// TIA Portal project "Servomotor" (V20)

(* hardware
DEVICE "S7-1500/ET200MP-Station_1"  S7-1500 station
   slot 0: "Profilschiene_0"  Rack  6ES7 590-1***0-0AA0
   slot 1: "PLC_1"  CPU 1515-2 PN  6ES7 515-2AM02-0AB0  V2.9
      slot 3: "CPU-Display_1"  6ES7591-1BA00-0AA0
      slot 32768: "PROFINET-Schnittstelle_1"  X1
         slot 32769: "Port_1"  X1 P1
         slot 32770: "Port_2"  X1 P2
      slot 33024: "PROFINET-Schnittstelle_2"  X2
         slot 33025: "Port_1"  X2 P1
      slot 34817: "Virtual CP interface port_1"  Virtual CP interface port  Virtual CP interface port
   slot 2: "AQ 8xU/I HS_1"  AQ 8xU/I HS  6ES7 532-5HF00-0AB0  V2.2
DEVICE "SINAMICS S_1"  SINAMICS S210
   slot 0: "Antriebsgerät_X"  S210 PN  6SL3210-5HB10-4xFx  V5.2.3
      slot 1: "PROFINET-Schnittstelle"  PROFINET
      slot 3: "Ethernet-IBN-Schnittstelle"  LAN
   slot 0: "Antriebsregelung"  S210 PN
      slot 200: "Power Module_1"  Antriebsregelung  6SL3210-5HB10-4xFx
      slot 300: "Geberauswertung_1"  Antriebsregelung  1FK2103-4AG0x-xDxx
      slot 400: "Messsystem_1"  Antriebsregelung  1FK2103-4AG0x-xDxx
      slot 1000: "Motor_1"  Antriebsregelung  1FK2103-4AG0x-xDxx
DEVICE "SINAMICS S_2"  SINAMICS S210
   slot 0: "Antriebsgerät_Y"  S210 PN  6SL3210-5HB10-4xFx  V5.2.3
      slot 1: "PROFINET-Schnittstelle"  PROFINET
      slot 3: "Ethernet-IBN-Schnittstelle"  LAN
   slot 0: "Antriebsregelung"  S210 PN
      slot 200: "Power Module_1"  Antriebsregelung  6SL3210-5HB10-4xFx
      slot 300: "Geberauswertung_1"  Antriebsregelung  1FK2103-4AG0x-xDxx
      slot 400: "Messsystem_1"  Antriebsregelung  1FK2103-4AG0x-xDxx
      slot 1000: "Motor_1"  Antriebsregelung  1FK2103-4AG0x-xDxx
DEVICE "SCALANCE X-200 IRT"  SCALANCE X-Station
   slot 0: "SCALANCE X-Rack"  Rail
   slot 0: "Switch_1"  SCALANCE X204 IRT  6GK5 204-0BA00-2BA3  V5.6
*)

// ===== PLC "PLC_1"  CPU 1515-2 PN =====

VAR_GLOBAL   // PLC tag table "Standard-Variablentabelle"
   "Tag_1" AT %AW30 : Int;
   "Tag_2" AT %AW32 : Int;
END_VAR

TYPE "typePOS_Axis"
   STRUCT
      Taster : Struct
         Power : Bool;
         Reset : Bool;
         Home : Bool;
         Halt : Bool;
         MoveAbsolute : Bool;
         MoveRelative : Bool;
         MoveVelocity : Bool;
         MoveJogForward : Bool;
         MoveJogBackward : Bool;
         Stop : Bool;
      END_STRUCT;
      Eingaben : Struct
         Absolutposition : LReal;
         Relativbewegung : LReal;
         Geschwindigkeit : LReal;
      END_STRUCT;
      Anzeigen : Struct
         TO_freigegeben : Bool;
         TO_referenziert : Bool;
         Sammelfehler : Bool;
         Done : Struct
            Power : Bool;
            Reset : Bool;
            Home : Bool;
            Halt : Bool;
            MoveAbsolute : Bool;
            MoveRelative : Bool;
            MoveVelocity : Bool;
            MoveJog : Bool;
            Stop : Bool;
         END_STRUCT;
         Busy : Struct
            Power : Bool;
            Reset : Bool;
            Home : Bool;
            Halt : Bool;
            MoveAbsolute : Bool;
            MoveRelative : Bool;
            MoveVelocity : Bool;
            MoveJog : Bool;
            Stop : Bool;
         END_STRUCT;
         CommandAborted : Struct
            Power : Bool;
            Reset : Bool;
            Home : Bool;
            Halt : Bool;
            MoveAbsolute : Bool;
            MoveRelative : Bool;
            MoveVelocity : Bool;
            MoveJog : Bool;
            Stop : Bool;
         END_STRUCT;
         Fehler : Struct
            Power : Bool;
            Reset : Bool;
            Home : Bool;
            Halt : Bool;
            MoveAbsolute : Bool;
            MoveRelative : Bool;
            MoveVelocity : Bool;
            MoveJog : Bool;
            Stop : Bool;
         END_STRUCT;
         Error_ID : Struct
            Power : Word;
            Reset : Word;
            Home : Word;
            Halt : Word;
            MoveAbsolute : Word;
            MoveRelative : Word;
            MoveVelocity : Word;
            MoveJog : Word;
            Stop : Word;
         END_STRUCT;
      END_STRUCT;
      Ausgaben : Struct
         Position : LReal;
         ActualPosition : LReal;
         ActualVelocity : LReal;
         ActualAcceleration : LReal;
      END_STRUCT;
   END_STRUCT;
END_TYPE

DATA_BLOCK "Daten"   // DB100
{ S7_Optimized_Access := 'TRUE' }
VERSION : 0.1
   VAR
      Daten_X_Achse : "typePOS_Axis";
      Daten_Y_Achse : "typePOS_Axis";
   END_VAR
BEGIN
END_DATA_BLOCK

DATA_BLOCK "IDB_Achse_X"   // DB101
{ S7_Optimized_Access := 'TRUE' }
VERSION : 0.1
// stored: InstanceOfName Achsensteuerung
"Achsensteuerung"
BEGIN
END_DATA_BLOCK

DATA_BLOCK "IDB_Achse_Y"   // DB102
{ S7_Optimized_Access := 'TRUE' }
VERSION : 0.1
// stored: InstanceOfName Achsensteuerung
"Achsensteuerung"
BEGIN
END_DATA_BLOCK

DATA_BLOCK "PositioningAxis_X"   // DB1, Motion_DB
{ S7_Optimized_Access := 'TRUE' }
AUTHOR : SIMATIC
FAMILY : MC_1500
VERSION : 6.0
// stored: InstanceOfName TO_PositioningAxis
"TO_PositioningAxis"
BEGIN
END_DATA_BLOCK

DATA_BLOCK "PositioningAxis_Y"   // DB2, Motion_DB
{ S7_Optimized_Access := 'TRUE' }
AUTHOR : SIMATIC
FAMILY : MC_1500
VERSION : 6.0
// stored: InstanceOfName TO_PositioningAxis
"TO_PositioningAxis"
BEGIN
END_DATA_BLOCK

FUNCTION_BLOCK "Achsensteuerung"   // FB101, FBD
{ S7_Optimized_Access := 'TRUE' }
VERSION : 0.1
   VAR_INPUT
      Achse : TO_PositioningAxis;
   END_VAR
   VAR_IN_OUT
      ioPOS_Axis : "typePOS_Axis";
   END_VAR
   VAR
      MDB_MC_POWER : MC_POWER;
      MDB_MC_RESET : MC_RESET;
      MDB_MC_MOVEABSOLUTE : MC_MOVEABSOLUTE;
      MDB_MC_HOME : MC_HOME;
      MDB_MC_HALT : MC_HALT;
      MD_MC_MOVERELATIVE : MC_MOVERELATIVE;
      MDB_MC_MOVEJOG : MC_MOVEJOG;
      MDB_MC_STOP : MC_STOP;
   END_VAR
BEGIN

REGION Network 1
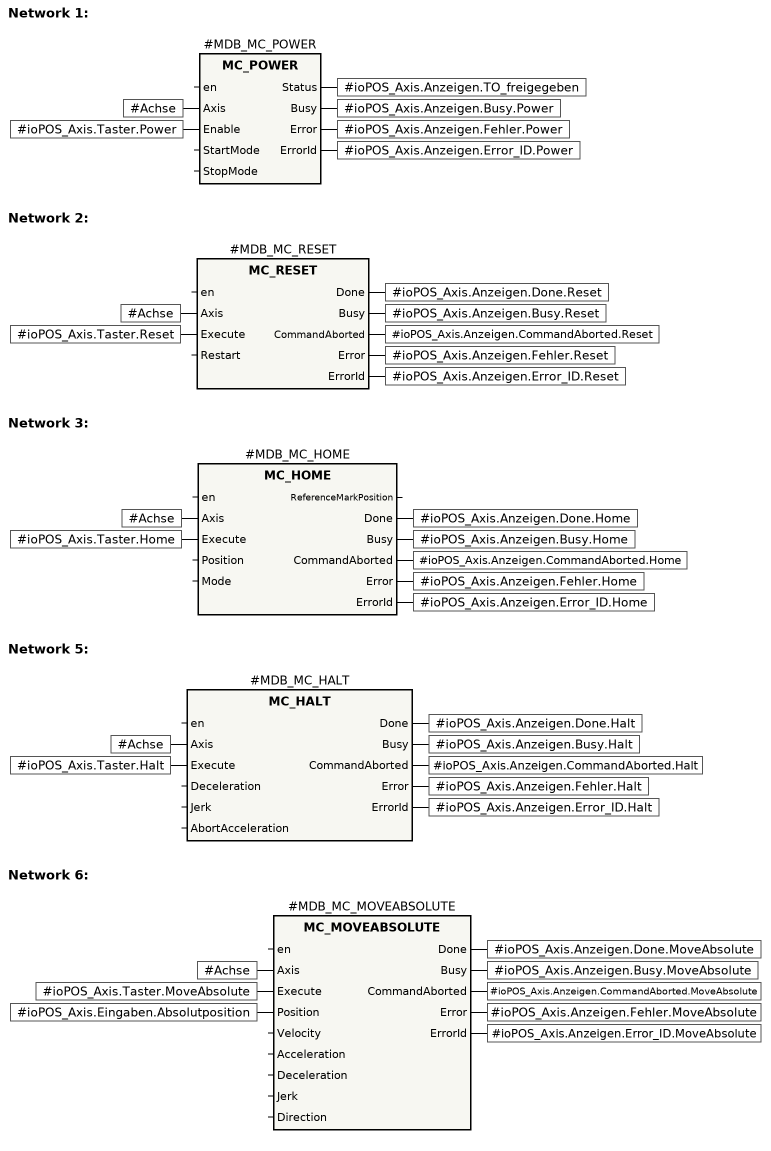
   #MDB_MC_POWER(Axis := #Achse,   // MC_POWER
                 Enable := #ioPOS_Axis.Taster.Power,
                 Status => #ioPOS_Axis.Anzeigen.TO_freigegeben,
                 Busy => #ioPOS_Axis.Anzeigen.Busy.Power,
                 Error => #ioPOS_Axis.Anzeigen.Fehler.Power,
                 ErrorId => #ioPOS_Axis.Anzeigen.Error_ID.Power);
END_REGION

REGION Network 2
   #MDB_MC_RESET(Axis := #Achse,   // MC_RESET
                 Execute := #ioPOS_Axis.Taster.Reset,
                 Done => #ioPOS_Axis.Anzeigen.Done.Reset,
                 Busy => #ioPOS_Axis.Anzeigen.Busy.Reset,
                 CommandAborted => #ioPOS_Axis.Anzeigen.CommandAborted.Reset,
                 Error => #ioPOS_Axis.Anzeigen.Fehler.Reset,
                 ErrorId => #ioPOS_Axis.Anzeigen.Error_ID.Reset);
END_REGION

REGION Network 3
   #MDB_MC_HOME(Axis := #Achse,   // MC_HOME
                Execute := #ioPOS_Axis.Taster.Home,
                Done => #ioPOS_Axis.Anzeigen.Done.Home,
                Busy => #ioPOS_Axis.Anzeigen.Busy.Home,
                CommandAborted => #ioPOS_Axis.Anzeigen.CommandAborted.Home,
                Error => #ioPOS_Axis.Anzeigen.Fehler.Home,
                ErrorId => #ioPOS_Axis.Anzeigen.Error_ID.Home);
END_REGION

REGION Network 4 (SCL)
   IF #ioPOS_Axis.Taster.Home
       AND #ioPOS_Axis.Anzeigen.Done.Home
       AND NOT #ioPOS_Axis.Anzeigen.Fehler.Home
   THEN
       #ioPOS_Axis.Anzeigen.TO_referenziert := TRUE;
   END_IF;
END_REGION

REGION Network 5
   #MDB_MC_HALT(Axis := #Achse,   // MC_HALT
                Execute := #ioPOS_Axis.Taster.Halt,
                Done => #ioPOS_Axis.Anzeigen.Done.Halt,
                Busy => #ioPOS_Axis.Anzeigen.Busy.Halt,
                CommandAborted => #ioPOS_Axis.Anzeigen.CommandAborted.Halt,
                Error => #ioPOS_Axis.Anzeigen.Fehler.Halt,
                ErrorId => #ioPOS_Axis.Anzeigen.Error_ID.Halt);
END_REGION

REGION Network 6
   #MDB_MC_MOVEABSOLUTE(Axis := #Achse,   // MC_MOVEABSOLUTE
                        Execute := #ioPOS_Axis.Taster.MoveAbsolute,
                        Position := #ioPOS_Axis.Eingaben.Absolutposition,
                        Done => #ioPOS_Axis.Anzeigen.Done.MoveAbsolute,
                        Busy => #ioPOS_Axis.Anzeigen.Busy.MoveAbsolute,
                        CommandAborted => #ioPOS_Axis.Anzeigen.CommandAborted.MoveAbsolute,
                        Error => #ioPOS_Axis.Anzeigen.Fehler.MoveAbsolute,
                        ErrorId => #ioPOS_Axis.Anzeigen.Error_ID.MoveAbsolute);
END_REGION

REGION Network 7 (SCL)
   #ioPOS_Axis.Ausgaben.Position := #Achse.Position;
   #ioPOS_Axis.Ausgaben.ActualPosition := #Achse.ActualPosition;
   #ioPOS_Axis.Ausgaben.ActualVelocity := #Achse.ActualVelocity;
   #ioPOS_Axis.Ausgaben.ActualAcceleration := #Achse.ActualAcceleration;
END_REGION

REGION Network 8
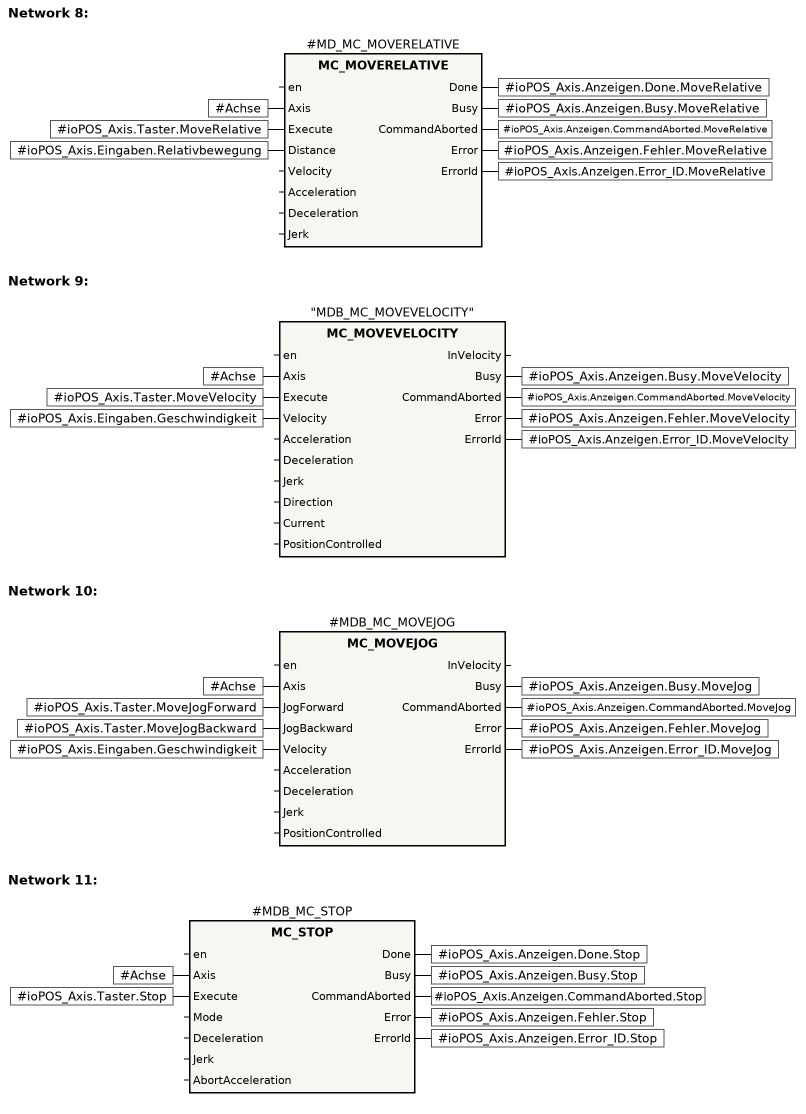
   #MD_MC_MOVERELATIVE(Axis := #Achse,   // MC_MOVERELATIVE
                       Execute := #ioPOS_Axis.Taster.MoveRelative,
                       Distance := #ioPOS_Axis.Eingaben.Relativbewegung,
                       Done => #ioPOS_Axis.Anzeigen.Done.MoveRelative,
                       Busy => #ioPOS_Axis.Anzeigen.Busy.MoveRelative,
                       CommandAborted => #ioPOS_Axis.Anzeigen.CommandAborted.MoveRelative,
                       Error => #ioPOS_Axis.Anzeigen.Fehler.MoveRelative,
                       ErrorId => #ioPOS_Axis.Anzeigen.Error_ID.MoveRelative);
END_REGION

REGION Network 9
   "MDB_MC_MOVEVELOCITY"(Axis := #Achse,   // MC_MOVEVELOCITY
                         Execute := #ioPOS_Axis.Taster.MoveVelocity,
                         Velocity := #ioPOS_Axis.Eingaben.Geschwindigkeit,
                         Busy => #ioPOS_Axis.Anzeigen.Busy.MoveVelocity,
                         CommandAborted => #ioPOS_Axis.Anzeigen.CommandAborted.MoveVelocity,
                         Error => #ioPOS_Axis.Anzeigen.Fehler.MoveVelocity,
                         ErrorId => #ioPOS_Axis.Anzeigen.Error_ID.MoveVelocity);
END_REGION

REGION Network 10
   #MDB_MC_MOVEJOG(Axis := #Achse,   // MC_MOVEJOG
                   JogForward := #ioPOS_Axis.Taster.MoveJogForward,
                   JogBackward := #ioPOS_Axis.Taster.MoveJogBackward,
                   Velocity := #ioPOS_Axis.Eingaben.Geschwindigkeit,
                   Busy => #ioPOS_Axis.Anzeigen.Busy.MoveJog,
                   CommandAborted => #ioPOS_Axis.Anzeigen.CommandAborted.MoveJog,
                   Error => #ioPOS_Axis.Anzeigen.Fehler.MoveJog,
                   ErrorId => #ioPOS_Axis.Anzeigen.Error_ID.MoveJog);
END_REGION

REGION Network 11
   #MDB_MC_STOP(Axis := #Achse,   // MC_STOP
                Execute := #ioPOS_Axis.Taster.Stop,
                Done => #ioPOS_Axis.Anzeigen.Done.Stop,
                Busy => #ioPOS_Axis.Anzeigen.Busy.Stop,
                CommandAborted => #ioPOS_Axis.Anzeigen.CommandAborted.Stop,
                Error => #ioPOS_Axis.Anzeigen.Fehler.Stop,
                ErrorId => #ioPOS_Axis.Anzeigen.Error_ID.Stop);
END_REGION

REGION Network 12 (SCL)
   // Sammelfehler
   #ioPOS_Axis.Anzeigen.Sammelfehler := #ioPOS_Axis.Anzeigen.Fehler.Power
                                       OR #ioPOS_Axis.Anzeigen.Fehler.Reset
                                       OR #ioPOS_Axis.Anzeigen.Fehler.Home
                                       OR #ioPOS_Axis.Anzeigen.Fehler.Halt
                                       OR #ioPOS_Axis.Anzeigen.Fehler.MoveAbsolute
                                       OR #ioPOS_Axis.Anzeigen.Fehler.MoveRelative
                                       OR #ioPOS_Axis.Anzeigen.Fehler.MoveVelocity
                                       OR #ioPOS_Axis.Anzeigen.Fehler.MoveJog
                                       OR #ioPOS_Axis.Anzeigen.Fehler.Stop;
END_REGION
END_FUNCTION_BLOCK

ORGANIZATION_BLOCK "Main"   // OB1, FBD, ProgramCycle
TITLE = "Main Program Sweep (Cycle)"
{ S7_Optimized_Access := 'TRUE' }
VERSION : 0.1
   VAR_INPUT
      Initial_Call : Bool;   // Initial call of this OB
      Remanence : Bool;   // =True, if remanent data are available
   END_VAR
   VAR_TEMP
      tmpNorm : LReal;
   END_VAR
BEGIN

REGION Network 1
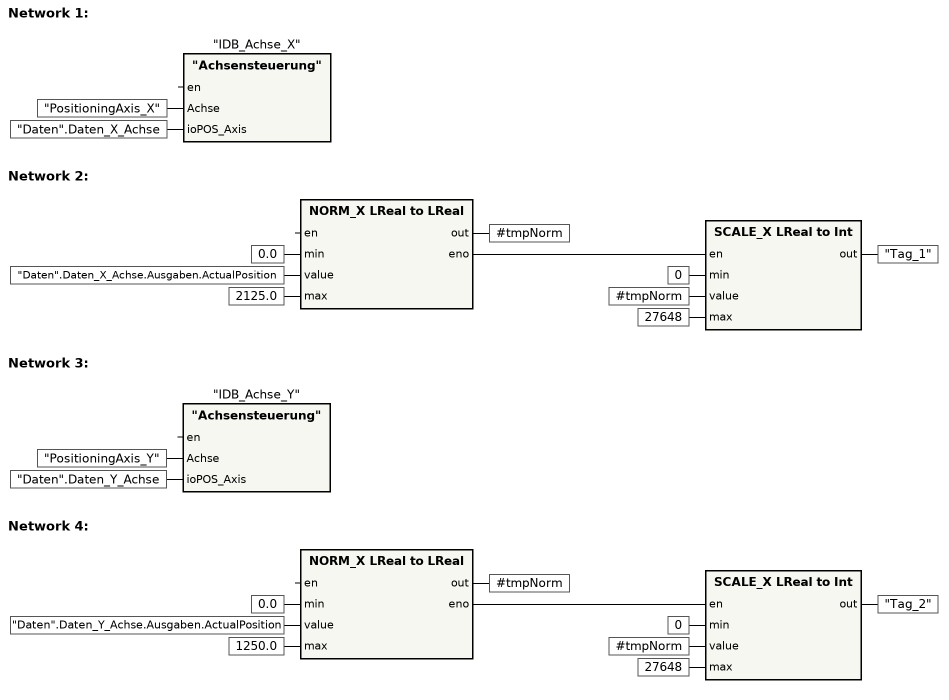
   "IDB_Achse_X"(Achse := "PositioningAxis_X", ioPOS_Axis := "Daten".Daten_X_Achse);   // "Achsensteuerung"
END_REGION

REGION Network 2
   #tmpNorm := NORM_X(MIN := 0.0, VALUE := "Daten".Daten_X_Achse.Ausgaben.ActualPosition, MAX := 2125.0);
   "Tag_1" := SCALE_X(MIN := 0, VALUE := #tmpNorm, MAX := 27648);
END_REGION

REGION Network 3
   "IDB_Achse_Y"(Achse := "PositioningAxis_Y", ioPOS_Axis := "Daten".Daten_Y_Achse);   // "Achsensteuerung"
END_REGION

REGION Network 4
   #tmpNorm := NORM_X(MIN := 0.0, VALUE := "Daten".Daten_Y_Achse.Ausgaben.ActualPosition, MAX := 1250.0);
   "Tag_2" := SCALE_X(MIN := 0, VALUE := #tmpNorm, MAX := 27648);
END_REGION
END_ORGANIZATION_BLOCK